// SIMATIC S7-200 SMART project (STEP 7-Micro/WIN SMART), CPU SR40

SYMBOL_TABLE 系统符号
Clock_1s         SM0.5    // 针对 1 s 的周期时间，时钟脉冲接通 0.5 s，断开 0.5 s.
END_SYMBOL_TABLE

ORGANIZATION_BLOCK MAIN:OB1
TITLE=程序注释
BEGIN
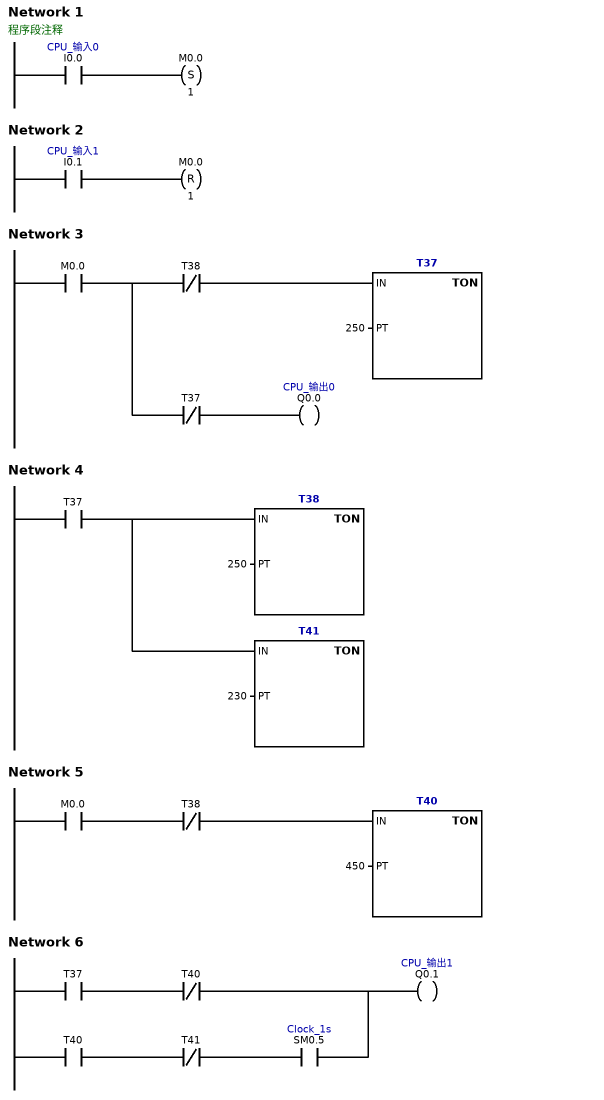
Network 1
// 程序段注释
LD     CPU_输入0:I0.0
S      M0.0, 1
Network 2
LD     CPU_输入1:I0.1
R      M0.0, 1
Network 3
LD     M0.0
LPS
AN     T38
TON    T37, 250
LPP
AN     T37
=      CPU_输出0:Q0.0
Network 4
LD     T37
TON    T38, 250
TON    T41, 230
Network 5
LD     M0.0
AN     T38
TON    T40, 450
Network 6
LD     T37
AN     T40
LD     T40
AN     T41
A      Clock_1s:SM0.5
OLD
=      CPU_输出1:Q0.1
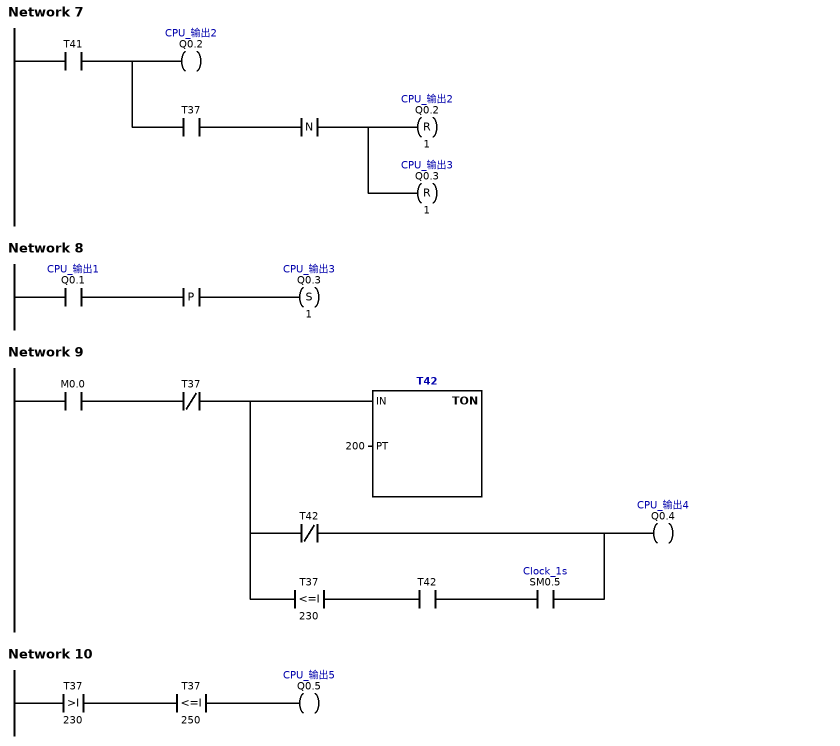
Network 7
LD     T41
=      CPU_输出2:Q0.2
A      T37
ED
R      CPU_输出2:Q0.2, 1
R      CPU_输出3:Q0.3, 1
Network 8
LD     CPU_输出1:Q0.1
EU
S      CPU_输出3:Q0.3, 1
Network 9
LD     M0.0
AN     T37
TON    T42, 200
LDN    T42
LDW<=  T37, 230
A      T42
A      Clock_1s:SM0.5
OLD
ALD
=      CPU_输出4:Q0.4
Network 10
LDW>   T37, 230
AW<=   T37, 250
=      CPU_输出5:Q0.5
END_ORGANIZATION_BLOCK
